{attribute addProperty BoxType "EM7004-0000-0017"}
{attribute addProperty Id "Output_0BIT10.1251Output_1BIT10.1252Output_2BIT10.1253Output_3BIT10.1254Output_4BIT10.1255Output_5BIT10.1256Output_6BIT10.1257Output_7BIT10.1258Output_8BIT10.1259Output_9BIT10.12510Output_10BIT10.12511Output_11BIT10.12512Output_12BIT10.12513Output_13BIT10.12514Output_14BIT10.12515Output_15BIT10.12516"}
{attribute addProperty CRC "3148183389"}
{attribute addProperty SizeInBites "16"}
{attribute addProperty SizeInBytes "2"}
TYPE Output_BBA5775D :
STRUCT
	{attribute addProperty Name "Output_0"}
	Output_0 : BIT;
	{attribute addProperty Name "Output_1"}
	Output_1 : BIT;
	{attribute addProperty Name "Output_2"}
	Output_2 : BIT;
	{attribute addProperty Name "Output_3"}
	Output_3 : BIT;
	{attribute addProperty Name "Output_4"}
	Output_4 : BIT;
	{attribute addProperty Name "Output_5"}
	Output_5 : BIT;
	{attribute addProperty Name "Output_6"}
	Output_6 : BIT;
	{attribute addProperty Name "Output_7"}
	Output_7 : BIT;
	{attribute addProperty Name "Output_8"}
	Output_8 : BIT;
	{attribute addProperty Name "Output_9"}
	Output_9 : BIT;
	{attribute addProperty Name "Output_10"}
	Output_10 : BIT;
	{attribute addProperty Name "Output_11"}
	Output_11 : BIT;
	{attribute addProperty Name "Output_12"}
	Output_12 : BIT;
	{attribute addProperty Name "Output_13"}
	Output_13 : BIT;
	{attribute addProperty Name "Output_14"}
	Output_14 : BIT;
	{attribute addProperty Name "Output_15"}
	Output_15 : BIT;
END_STRUCT
END_TYPE

(* stored: Version 1.2.0.0, ProductVersion 3.1.4024.9
   DUT Output_BBA5775D: Id {ba59ce86-b032-463c-984b-c64eddc166b1} *)
